FUNCTION F_StringLength : UDINT
VAR_IN_OUT CONSTANT
	str : STRING;
END_VAR
VAR
	pByte : POINTER TO BYTE;
END_VAR

pByte := ADR(str);

WHILE pByte^ <> 0 DO
	pByte := pByte + 1;
	F_StringLength := F_StringLength + 1;
END_WHILE

END_FUNCTION

(* stored: Version 1.1.0.1, ProductVersion 3.1.4024.15
   POU F_StringLength: Id {89a0ba35-a760-468f-89a1-46b54b1d6306}, SpecialFunc None *)
